FUNCTION_BLOCK QUERY_STATION3
  {SET_ATTRIBUTE(OpcUa, SERVICE)}
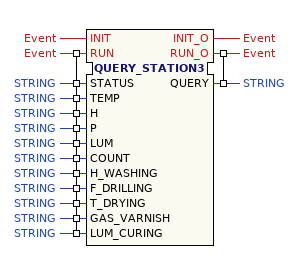
  EVENT_INPUT
    INIT;
    RUN WITH STATUS, TEMP, H, P, LUM, COUNT, H_WASHING, F_DRILLING, T_DRYING, GAS_VARNISH, LUM_CURING; {SET_ATTRIBUTE(OpcUa, Method)}
  END_EVENT
  EVENT_OUTPUT
    INIT_O;
    RUN_O WITH QUERY;
  END_EVENT
  VAR_INPUT
    STATUS : STRING;
    TEMP : STRING;
    H : STRING;
    P : STRING;
    LUM : STRING;
    COUNT : STRING;
    H_WASHING : STRING;
    F_DRILLING : STRING;
    T_DRYING : STRING;
    GAS_VARNISH : STRING;
    LUM_CURING : STRING;
  END_VAR
  VAR_OUTPUT
    QUERY : STRING;
  END_VAR
END_FUNCTION_BLOCK
